FUNCTION_BLOCK CMP_OC_DW
VAR_INPUT
	BOOL_INTERLOCK : BOOL; (*INTERLOCK*)
	DWORD_1: DWORD;		(*WORD 1*)
	END_VAR


VAR_OUTPUT
	BZ_OUTPUT_BOOL : BOOL;
END_VAR


VAR
	OUT_1: BOOL;
END_VAR

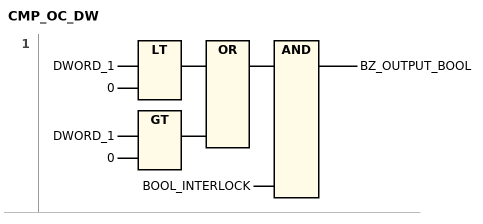
// NETWORK 1
BZ_OUTPUT_BOOL := (DWORD_1 < 0 OR DWORD_1 > 0) AND BOOL_INTERLOCK;

END_FUNCTION_BLOCK

(* stored: Version 1.1.0.1, ProductVersion 3.1.4024.12
   POU CMP_OC_DW: Id {13a7039e-d774-49e4-9042-02adfb58cf9c}, SpecialFunc None *)
